(* Logix 5000 project; controller ECE4350_Experiment3 vendor 1 type 14 code 3 rev 13.1; software revision 13.03 *)
// Engineers:
// Angelino Lefevers
// Jacob Little

TASK MainTask (continuous, watchdog 500 ms) : MainProgram

MODULES
   Local : vendor 1 type 14 code 3 (ICP 0, rev 13.1)
       : 1756-IB16 (ICP 2, rev 2.1, Input RPI 10 ms)
       : vendor 1 type 7 code 18 (ICP 4, rev 1.1, Output RPI 10 ms)
END_MODULES

PROGRAM MainProgram   (* routine attr 65 MainRoutine *)
VAR
   CT1 : COUNTER := (PRE := 3);   // Counter 1
   FM1 : ALIAS FOR Local:4:O.Data.2;   // Fan Motor 1
   GL1 : ALIAS FOR Local:4:O.Data.0;   // Green LED 1
   LAL : ALIAS FOR Local:4:O.Data.3;   // Actuator - Right to Left
   LAR : ALIAS FOR Local:4:O.Data.4;   // Actuator - Left to Right (LAL Must be activated as well)
   LS1 : ALIAS FOR Local:2:I.Data.3;   // Right Stop for L.A.
   LS2 : ALIAS FOR Local:2:I.Data.2;   // Left Stop for L.A.
   ONS1 : BOOL;   // one shot for solenoid
   ONS10 : BOOL;   // one shot
   ONS2 : BOOL;   // one shot
   ONS3 : BOOL;   // one shot
   ONS4 : BOOL;   // one shot
   ONS5 : BOOL;   // one shot
   ONS6 : BOOL;   // one shot
   ONS7 : BOOL;   // one shot
   ONS8 : BOOL;   // one shot
   ONS9 : BOOL;   // one shot
   PB1 : ALIAS FOR Local:2:I.Data.0;   // Push Button 1
   PB2 : ALIAS FOR Local:2:I.Data.1;   // Push Button 2 Returns L.A. to left stop
   PS1 : ALIAS FOR Local:2:I.Data.4;   // Photo Switch 1
   RL1 : ALIAS FOR Local:4:O.Data.1;   // Red LED 1
   RS1 : ALIAS FOR Local:2:I.Data.6;   // Reed Switch 1
   SL1 : ALIAS FOR Local:4:O.Data.5;   // Solenoid
   TM1 : TIMER := (PRE := 5000);   // Timer 1 PB1 5 Second Timer
   TM2 : TIMER := (PRE := 10000);   // Timer 2
   TP1 : ALIAS FOR Local:2:I.Data.5;   // Temperature Switch 1
END_VAR

ROUTINE MainRoutine   (* ladder *)
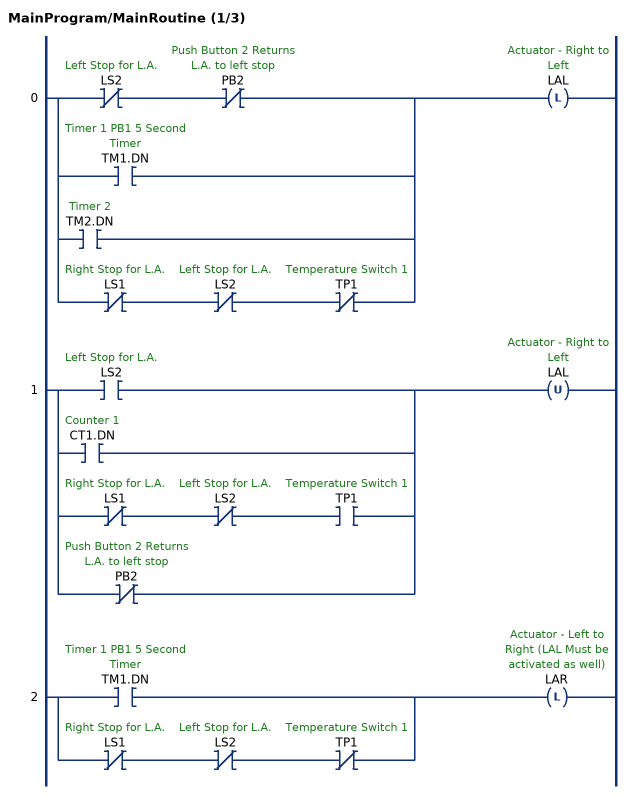
   0: [XIO(LS2) XIO(PB2) ,XIC(TM1.DN) ,XIC(TM2.DN) ,XIO(LS1) XIO(LS2) XIO(TP1) ]OTL(LAL);
   1: [XIC(LS2) ,XIC(CT1.DN) ,XIO(LS1) XIO(LS2) XIC(TP1) ,XIO(PB2) ]OTU(LAL);
   2: [XIC(TM1.DN) ,XIO(LS1) XIO(LS2) XIO(TP1) ]OTL(LAR);
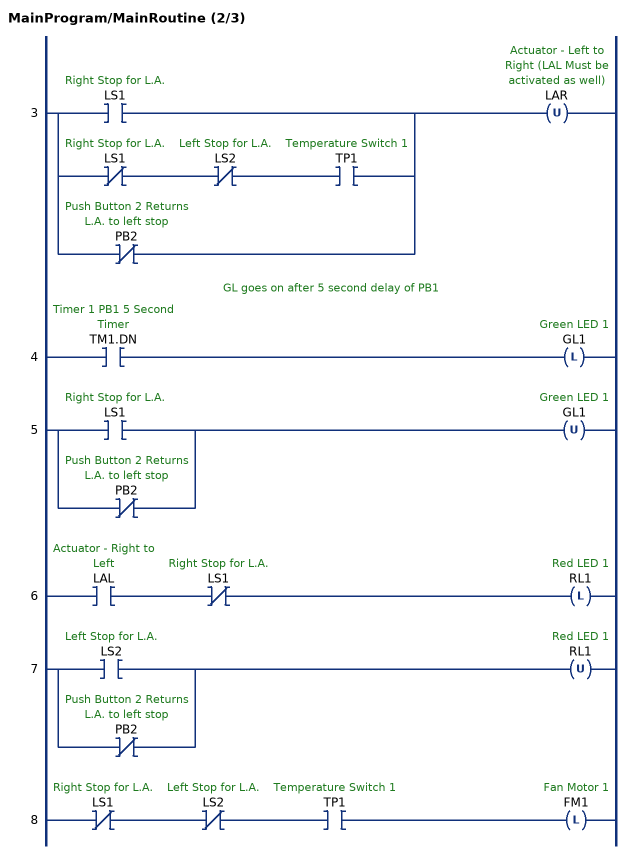
   3: [XIC(LS1) ,XIO(LS1) XIO(LS2) XIC(TP1) ,XIO(PB2) ]OTU(LAR);
   // GL goes on after 5 second delay of PB1
   4: XIC(TM1.DN)OTL(GL1);
   5: [XIC(LS1) ,XIO(PB2) ]OTU(GL1);
   6: XIC(LAL)XIO(LS1)OTL(RL1);
   7: [XIC(LS2) ,XIO(PB2) ]OTU(RL1);
   8: XIO(LS1)XIO(LS2)XIC(TP1)OTL(FM1);
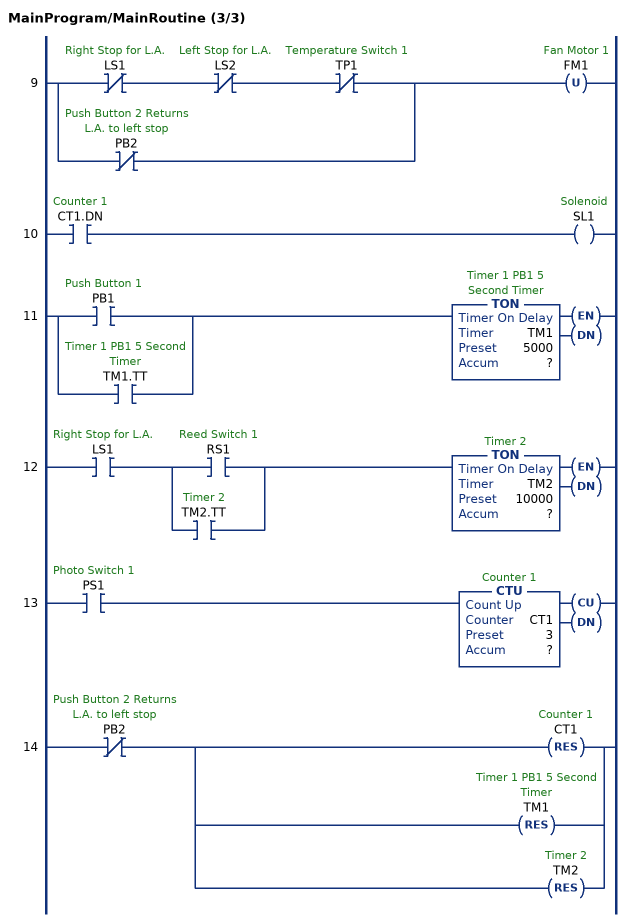
   9: [XIO(LS1) XIO(LS2) XIO(TP1) ,XIO(PB2) ]OTU(FM1);
   10: XIC(CT1.DN)OTE(SL1);
   11: [XIC(PB1) ,XIC(TM1.TT) ]TON(TM1,?,?);
   12: XIC(LS1)[XIC(RS1) ,XIC(TM2.TT) ]TON(TM2,?,?);
   13: XIC(PS1)CTU(CT1,?,?);
   14: XIO(PB2)[RES(CT1) ,RES(TM1) ,RES(TM2) ];
END_ROUTINE
END_PROGRAM
